{attribute addProperty BoxType "EJ2521-0224-0016"}
{attribute addProperty Id "Enable_PLSBIT10.1251OutputBIT10.1254"}
{attribute addProperty CRC "90070654"}
{attribute addProperty SizeInBites "16"}
{attribute addProperty SizeInBytes "2"}
TYPE Control_055E5E7E :
STRUCT
	{attribute addProperty Name "Enable_PLS"}
	Enable_PLS : BOOL;
	{attribute 'hide'}
	reserve_1_BIT_0 : BOOL;
	{attribute 'hide'}
	reserve_1_BIT_1 : BOOL;
	{attribute addProperty Name "Output"}
	Output : BOOL;
	{attribute 'hide'}
	reserve_2_BIT_0 : BOOL;
	{attribute 'hide'}
	reserve_2_BIT_1 : BOOL;
	{attribute 'hide'}
	reserve_2_BIT_2 : BOOL;
	{attribute 'hide'}
	reserve_2_BIT_3 : BOOL;
	{attribute 'hide'}
	reserve_3 : BYTE;
END_STRUCT
END_TYPE

(* stored: Version 1.2.0.0, ProductVersion 3.1.4024.9
   DUT Control_055E5E7E: Id {ecc6726d-6a5c-43f1-9f66-e72ab184405e} *)
